(* PLC project InterlockTest *)
(* stored: creationDateTime 2024-01-01T00:00:00, modificationDateTime 2024-01-01T00:00:00 *)

PROGRAM Main
  VAR
    X001 : BOOL;
    X002 : BOOL;
    Y001 : BOOL;
    Y002 : BOOL;
  END_VAR

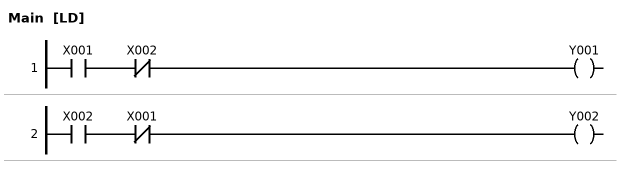
(* LD diagram, written out as Structured Text *)
Y001 := X001 AND NOT X002;
Y002 := X002 AND NOT X001;
END_PROGRAM

CONFIGURATION Config
  RESOURCE Res ON PLC
    TASK Main(INTERVAL := T#20ms, PRIORITY := 0);
    PROGRAM Main WITH Main : Main;
  END_RESOURCE
END_CONFIGURATION
